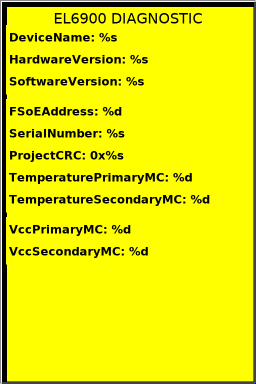
VISUALIZATION V_PH_EL6900_DIAG  // 256x384
VAR_INPUT
	stEL6900DiagnosticData		:ST_EL6900_DiagnosticData;
END_VAR
    Rectangle (2,2 256x384), colour toggle: stEL6900DiagnosticData.bGeneralError
    Label (5,6 246x25), "EL6900 DIAGNOSTIC"
    Rectangle (6,25 242x25), "DeviceName: %s", text variable: stEL6900DiagnosticData.sDeviceName
    Rectangle (6,47 242x25), "HardwareVersion: %s", text variable: stEL6900DiagnosticData.sHardwareVersion
    Rectangle (6,69 242x25), "SoftwareVersion: %s", text variable: stEL6900DiagnosticData.sSoftwareVersion
    Rectangle (6,121 242x25), "SerialNumber: %s", text variable: stEL6900DiagnosticData.sSerialNumber
    Rectangle (6,143 242x25), "ProjectCRC: 0x%s", text variable: stEL6900DiagnosticData.sProjectCRC
    Rectangle (6,187 242x25), "TemperatureSecondaryMC: %d", text variable: stEL6900DiagnosticData.wTemperatureSecondaryMC
    Rectangle (6,99 242x25), "FSoEAddress: %d", text variable: stEL6900DiagnosticData.dwFSoEAddress
    Rectangle (6,165 242x25), "TemperaturePrimaryMC: %d", text variable: stEL6900DiagnosticData.wTemperaturePrimaryMC
    Rectangle (6,217 242x25), "VccPrimaryMC: %d", text variable: stEL6900DiagnosticData.wVccPrimaryMC
    Rectangle (6,239 242x25), "VccSecondaryMC: %d", text variable: stEL6900DiagnosticData.wVccSecondaryMC
END_VISUALIZATION

(* stored: Version 1.1.0.1, ProductVersion 3.1.4024.4
   Visu V_PH_EL6900_DIAG: Id {9649e7a9-d4a5-4a5e-80de-ff27aa8f19b5} *)
